// TwinCAT 3 PLC project PLC
// ProgramVersion: 3.1.4023.0
// libraries:
//   Tc2_MC2, * (Beckhoff Automation GmbH)
//   Tc2_Standard, * (Beckhoff Automation GmbH)
//   Tc2_System, * (Beckhoff Automation GmbH)
//   Tc3_MC2_AdvancedHoming, * (Beckhoff Automation GmbH)
//   Tc3_Module, * (Beckhoff Automation GmbH)
// project tree:
//   DUTs/Motion/ E_AxisParameters.TcTLEO, E_EncoderTypeClass.TcDUT, E_HomeSwitchTypeClass.TcDUT, E_HomingRoutines.TcTLEO, E_MotionFunctions.TcDUT, E_MotorTypeClass.TcDUT, E_RestorePosition.TcDUT, ST_AxisConfig.TcDUT, ST_AxisControl.TcDUT, ST_AxisDescription.TcDUT, ST_AxisError.TcDUT, ST_AxisInputs.TcDUT, ST_AxisPersistent.TcDUT, ST_AxisStatus.TcDUT, ST_AxisStruct.TcDUT, ST_GearAxis.TcDUT
//   GVLs/ GVL_APP.TcGVL, GVL.TcGVL
//   / PlcTask.TcTTO
//   POUs/ MAIN.TcPOU
//   POUs/Motion/ FB_Axis.TcPOU
//   POUs/Motion/Homing/ FB_Homing.TcPOU
// real-time tasks:
//   TASK PlcTask: cycle T#10ms, priority 20, ADS port 350
// motion (NC):
//   TASK NC-Task 1 SAF: cycle T#2ms, priority 4, ADS port 501
//   TASK NC-Task 1 SVB: cycle T#10ms, priority 8, ADS port 511
//   AXIS R1_Axis01_X1 (id 1)
//     OtherSettings: AllowMotionCmdToSlave=true
//     encoder EncType=1
//     drive DrvType=5
//       Analog: TorqueSetpointScale=10, ScaleFactorActTorque=0.1
//     controller CtrType=1
//       CtrPara: PriorControlFactor=1
//         Observer: BandWidth=20
//   AXIS R1_Axis02_X2 (id 2)
//     OtherSettings: AllowMotionCmdToSlave=true
//     encoder EncType=1
//     drive DrvType=5
//       Analog: TorqueSetpointScale=10, ScaleFactorActTorque=0.1
//     controller CtrType=1
//       CtrPara: PriorControlFactor=1
//         Observer: BandWidth=20
//   AXIS R1_Axis03_Y (id 3)
//     OtherSettings: AllowMotionCmdToSlave=true
//     encoder EncType=1
//     drive DrvType=5
//       Analog: TorqueSetpointScale=10, ScaleFactorActTorque=0.1
//     controller CtrType=1
//       CtrPara: PriorControlFactor=1
//         Observer: BandWidth=20
//   AXIS R1_Axis04_Z (id 4)
//     OtherSettings: AllowMotionCmdToSlave=true
//     encoder EncType=1
//     drive DrvType=5
//       Analog: TorqueSetpointScale=10, ScaleFactorActTorque=0.1
//     controller CtrType=1
//       CtrPara: PriorControlFactor=1
//         Observer: BandWidth=20
// variable links:
//   PLC/PLC Instance <-> NC-Task 1 SAF/Axes/R1_Axis01_X1
//     PlcTask Inputs/GVL.astAxes[1].Axis.NcToPlc <-> Outputs/ToPlc
//     PlcTask Outputs/GVL.astAxes[1].Axis.PlcToNc <-> Inputs/FromPlc
//   PLC/PLC Instance <-> NC-Task 1 SAF/Axes/R1_Axis02_X2
//     PlcTask Inputs/GVL.astAxes[2].Axis.NcToPlc <-> Outputs/ToPlc
//     PlcTask Outputs/GVL.astAxes[2].Axis.PlcToNc <-> Inputs/FromPlc
//   PLC/PLC Instance <-> NC-Task 1 SAF/Axes/R1_Axis03_Y
//     PlcTask Inputs/GVL.astAxes[3].Axis.NcToPlc <-> Outputs/ToPlc
//     PlcTask Outputs/GVL.astAxes[3].Axis.PlcToNc <-> Inputs/FromPlc
//   PLC/PLC Instance <-> NC-Task 1 SAF/Axes/R1_Axis04_Z
//     PlcTask Inputs/GVL.astAxes[4].Axis.NcToPlc <-> Outputs/ToPlc
//     PlcTask Outputs/GVL.astAxes[4].Axis.PlcToNc <-> Inputs/FromPlc

CONFIGURATION PLC
    RESOURCE PLC ON TwinCAT3
        TASK PlcTask(INTERVAL := T#10ms, PRIORITY := 20);
        PROGRAM MAIN WITH PlcTask : MAIN;
    END_RESOURCE
END_CONFIGURATION

// ---- DUTs/Motion/E_AxisParameters.TcTLEO
{attribute 'qualified_only'}
{attribute 'strict'}
TYPE E_AxisParameters :
(
//PLCopen specific parameters Index-Group 0x4000 + ID
    CommandedPosition := 1, //lreal taken from NcToPlc
    SWLimitForward := 2, //lreal IndexOffset= 16#0001_000E
    SWLimitBackward := 3, //lreal IndexOffset= 16#0001_000D
    EnableLimitForward := 4, //bool IndexOffset= 16#0001_000C
    EnableLimitBackward := 5, //bool IndexOffset= 16#0001_000B
    EnablePositionLagMonitoring := 6, //bool IndexOffset= 16#0002_0010
    MaxPositionLag := 7, //lreal IndexOffset= 16#0002_0012
    AxisMaxVelocity := 8, //lreal IndexOffset= 16#0000_0027
    ActualVelocity := 10, //lreal taken from NcToPlc
    CommandedVelocity := 11, //lreal taken from NcToPlc
    AxisDefaultAcceleration := 12, //lreal IndexOffset= 16#0000_0101
    AxisDefaultDeceleration := 14, //lreal IndexOffset= 16#0000_0102
    AxisDefaultJerk := 16, //lreal IndexOffset= 16#0000_0103

//Beckhoff specific parameters Index-Group 0x4000 + ID
    AxisId := 1000, //lreal IndexOffset= 16#0000_0001
    AxisManualVelocitySlow := 1001, //lreal IndexOffset= 16#0000_0008
    AxisManualVelocityFast := 1002, //lreal IndexOffset= 16#0000_0009
    AxisAccMax := 1004, //lreal IndexOffset= 16#0000_0101
    AxisDecMax := 1005, //lreal IndexOffset= 16#0000_0102
    AxisRapidTraverseVelocity := 1009, //lreal IndexOffset= 16#0000_000A
    AxisVelocityToCam := 1012, //lreal IndexOffset= 16#0000_0006
    AxisVelocityFromCam := 1013, //lreal IndexOffset= 16#0000_0007
    AxisJogIncrementForward := 1014, //lreal IndexOffset= 16#0000_0018
    AxisJogIncrementBackward := 1015, //lreal IndexOffset= 16#0000_0019
    MaxPositionLagFilterTime := 1022, //lreal IndexOffset= 16#0002_0013
    AxisEnPositionRangeMonitoring := 1023, //bool IndexOffset= 16#0000_000F
    AxisPositionRangeWindow := 1024, //lreal IndexOffset= 16#0000_0010
    AxisEnTargetPositionMonitoring:= 1025, //bool IndexOffset= 16#0000_0015
    AxisTargetPositionWindow := 1026, //lreal IndexOffset= 16#0000_0016
    AxisTargetPositionMonitoringTime := 1027, //lreal IndexOffset= 16#0000_0017
    AxisEnInTargetTimeout := 1028, //bool IndexOffset= 16#0000_0029
    AxisInTargetTimeout := 1029, //lreal IndexOffset= 16#0000_002A
    AxisEnMotionMonitoring := 1030, //bool IndexOffset= 16#0000_0011
    AxisMotionMonitoringWindow := 1031, //lreal IndexOffset= 16#0000_0028
    AxisMotionMonitoringTime := 1032, //lreal IndexOffset= 16#0000_0012
    AxisDelayTimeVeloPosition := 1033, //lreal IndexOffset= 16#0000_0104
    AxisEnLoopingDistance := 1034, //bool IndexOffset= 16#0000_0013
    AxisLoopingDistance := 1035, //lreal IndexOffset= 16#0000_0014
    AxisEnBacklashCompensation := 1036, //bool IndexOffset= 16#0000_002B
    AxisBacklash := 1037, //lreal IndexOffset= 16#0000_002C
    AxisEnDataPersistence := 1038, //bool IndexOffset= 16#0000_0030
    AxisRefVeloOnRefOutput := 1039, //lreal IndexOffset= 16#0003_0101
    AxisOverrideType := 1040, //lreal IndexOffset= 16#0000_0105
    //new since 4/2007
    AxisEncoderOffset := 1042, //lreal IndexOffset= 16#0001_0007
    AxisEncoderDirectionInverse := 1043, //bool IndexOffset= 16#0001_0008
    AxisEncoderMask := 1044, //dword IndexOffset= 16#0001_0015
    AxisEncoderModuloValue := 1045, //lreal IndexOffset= 16#0001_0009
    AxisModuloToleranceWindow := 1046, //lreal IndexOffset= 16#0001_001B
    AxisEnablePosCorrection := 1047, //bool IndexOffset= 16#0001_0016
    AxisPosCorrectionFilterTime := 1048, //lreal IndexOffset= 16#0001_0017
    //new since 1/2010
    AxisUnitInterpretation := 1049, //lreal IndexOffset= 16#0000_0026
    AxisMotorDirectionInverse := 1050, //bool  IndexOffset= 16#0003_0006
    //new since 1/2011
    AxisCycleTime := 1051, //lreal IndexOffset= 16#0000_0004
    //new since 5/2011
    AxisFastStopSignalType := 1052, //dword IndexOffset= 16#0000_001E
    AxisFastAcc := 1053, //lreal IndexOffset= 16#0000_010A
    AxisFastDec := 1054, //lreal IndexOffset= 16#0000_010B
    AxisFastJerk := 1055, //lreal IndexOffset= 16#0000_010C
    // new since 1/2012 *)
    AxisEncoderScalingNumerator := 1056, //lreal IndexOffset= 16#0001_0023 - available in Tc3
    AxisEncoderScalingDenominator := 1057, //lreal IndexOffset= 16#0001_0024 - available in Tc3
    (* new since 7/2016 *)
    AxisVeloJumpFactor := 1060, //lreal IndexOffset= 16#0000_0106
    AxisToleranceBallAuxAxis := 1061, //lreal IndexOffset= 16#0000_0108
    AxisMaxPositionDeviationAuxAxis := 1062, //lreal IndexOffset= 16#0000_0109
    AxisErrorPropagationMode := 1063, //dword IndexOffset= 16#0000_001A
    AxisErrorPropagationDelay := 1064, //lreal IndexOffset= 16#0000_001B
    AxisCoupleSlaveToActualValues := 1065, //bool IndexOffset= 16#0000_001C
    AxisAllowMotionCmdToSlaveAxis := 1066, //bool IndexOffset= 16#0000_0020
    AxisAllowMotionCmdToExtSetAxis := 1067, //bool IndexOffset= 16#0000_0021
    AxisEncoderSubMask := 1068, //dword IndexOffset= 16#0001_0108
    AxisEncoderReferenceSystem := 1069, //dword IndexOffset= 16#0001_0019
    AxisEncoderPositionFilterPT1 := 1070, //lreal IndexOffset= 16#0001_0010
    AxisEncoderVelocityFilterPT1 := 1071, //lreal IndexOffset= 16#0001_0011
    AxisEncoderAccelerationFilterPT1 := 1072, //lreal IndexOffset= 16#0001_0012
    AxisEncoderMode := 1073, //dword IndexOffset= 16#0001_000A
    AxisEncoderHomingInvDirCamSearch := 1074, //bool IndexOffset= 16#0001_0101
    AxisEncoderHomingInvDirSyncSearch := 1075, //bool IndexOffset= 16#0001_0102
    AxisEncoderHomingCalibValue := 1076, //lreal IndexOffset= 16#0001_0103
    AxisEncoderReferenceMode := 1077, //dword IndexOffset= 16#0001_0107
    AxisRefVeloOutputRatio := 1078, //lreal IndexOffset= 16#0003_0102
    AxisDrivePositionOutputScaling := 1079, //lreal IndexOffset= 16#0003_0109
    AxisDriveVelocityOutputScaling := 1080, //lreal IndexOffset= 16#0003_0105
    AxisDriveVelocityOutputDelay := 1081, //lreal IndexOffset= 16#0003_010D
    AxisDriveMinOutputLimitation := 1082, //lreal IndexOffset= 16#0003_000B
    AxisDriveMaxOutputLimitation := 1083, //lreal IndexOffset= 16#0003_000C
    AxisTorqueInputScaling := 1084, //lreal IndexOffset= 16#0003_0031 - available in Tc3
    AxisTorqueInputFilterPT1 := 1085, //lreal IndexOffset= 16#0003_0032 - available in Tc3
    AxisTorqueDerivationInputFilterPT1 := 1086, //lreal IndexOffset= 16#0003_0033 - available in Tc3
    AxisTorqueOutputScaling := 1087, //lreal IndexOffset= 16#0003_010B
    AxisTorqueOutputDelay := 1088, //lreal IndexOffset= 16#0003_010F
    AxisAccelerationOutputScaling := 1089, //lreal IndexOffset= 16#0003_010A
    AxisAccelerationOutputDelay := 1090, //lreal IndexOffset= 16#0003_010E
    AxisDrivePositionOutputSmoothFilterType := 1091, //dword IndexOffset= 16#0003_0110
    AxisDrivePositionOutputSmoothFilterTime := 1092, //lreal IndexOffset= 16#0003_0111
    AxisDrivePositionOutputSmoothFilterOrder := 1093, //dword IndexOffset= 16#0003_0112
    AxisDriveMode := 1094, //dword IndexOffset= 16#0003_000A
    AxisDriftCompensationOffset := 1095, //lreal IndexOffset= 16#0003_0104
    AxisPositionControlKv := 1096, //lreal IndexOffset= 16#0002_0102
    AxisCtrlVelocityPreCtrlWeight := 1097, //lreal IndexOffset= 16#0002_000B
    AxisControllerMode := 1098, //dword IndexOffset= 16#0002_000A
    AxisCtrlAutoOffset := 1099, //bool IndexOffset= 16#0002_0110
    AxisCtrlAutoOffsetTimer := 1100, //lreal IndexOffset= 16#0002_0115
    AxisCtrlAutoOffsetLimit := 1101, //lreal IndexOffset= 16#0002_0114
    AxisSlaveCouplingControlKcp := 1102, //lreal IndexOffset= 16#0002_010F
    AxisCtrlOutputLimit := 1103, //lreal IndexOffset= 16#0002_0100

//Beckhoff specific axis status information - READ ONLY Index-Group 0x4100 + ID
    AxisTargetPosition := 2000, //lreal IndexOffset= 16#0000_0013
    AxisRemainingTimeToGo := 2001, //lreal IndexOffset= 16#0000_0014
    AxisRemainingDistanceToGo := 2002, //lreal IndexOffset= 16#0000_0022, 16#0000_0042

//Beckhoff specific axis functions
    //read/write gear ratio of a slave
    AxisGearRatio := 3000, //lreal read: IndexGroup=0x4100+ID, IdxOffset=16#0000_0022,
                                 //write:IndexGroup=0x4200+ID, IdxOffset=16#0000_0042

//Beckhoff specific other parameters
    //new since 1/2011
    NcSafCycleTime := 4000, //lreal IndexOffset= 16#0000_0010
    NcSvbCycleTime := 4001 //lreal IndexOffset= 16#0000_0012

);
END_TYPE

// ---- DUTs/Motion/E_EncoderTypeClass.TcDUT
TYPE E_EncoderTypeClass :
(
    eNoEncoder := 0,
    eIncrementalEncoder := 1,
    eAbsoluteEncoder := 2
) := eNoEncoder;
END_TYPE

// ---- DUTs/Motion/E_HomeSwitchTypeClass.TcDUT
TYPE E_HomeSwitchTypeClass:
(
    eNoSwitch := 0, //no physical switch for homing present
    eHomeSwitchPresent := 1, //dedicated homing switch present
    eUseBwdLimit := 2, //Bwd limit switch is used as a homing switch
    eUseFwdLimit := 3 //Fwd limit switch is used as a homing switch
) := eNoSwitch;
END_TYPE

// ---- DUTs/Motion/E_HomingRoutines.TcTLEO
{attribute 'qualified_only'}
{attribute 'strict'}
TYPE E_HomingRoutines :
(
    eNoHoming := 0,

    //0X: LIMIT Switch
    //Home to bBwdLimit, record position on first approach
    eHomeToLimit_Bwd := 1,
    //Home to bFwdLimit, record position on first approach
    eHomeToLimit_Fwd := 2,
    //Find bBwdLimit (using towardsCam speed), then reverse direction looking FOR falling edge (using fromCam speed)
    //eHomeToLimit_Bwd_2Speeds := 3,
    //Find bFwdLimit (using towardsCam speed), then reverse direction looking for falling edge (using fromCam speed)
    //eHomeToLimit_Fwd_2Speeds := 4,

    //1X: Home Sensor
    //Home to bHome in Bwd direction (will reverse direction if limit hit), record position on first approach
    eHomeToRef_Bwd := 11,
    //Home to bHome in Fwd direction (will reverse direction if limit hit), record position on first approach
    eHomeToRef_Fwd := 12,
    //Find bHome in Bwd direction (using towardsCam speed) then reverse direction looking for falling edge (using fromCam speed), will reverse direction if limit hit
    //eHomeToRef_Bwd_2Speeds := 13,
    //Find bHome in Fwd direction (using towardsCam speed) then reverse direction looking for falling edge (using fromCam speed), will reverse direction if limit hit
    //eHomeToRef_Fwd_2Speeds := 14,

    //2X: Enc Pulse
    //Home to EncRefPulse in Bwd direction (used for single turn rotary axis without limit switches)
    eHomeToEncPulse_Bwd := 21,
    //Home to EncRefPulse in Fwd direction (used for single turn rotary axis without limit switches)
    eHomeToEncPulse_Fwd := 22,
    //Home to EncRefPulse via bBwdLimit (using towardsCam speed), then reverse direction looking for falling edge on ref pulse (using fromCam speed)
    eHomeToEncPulse_viaBwdLimit := 23,
    //Home to EncRefPulse via bFwdLimit (using towardsCam speed), then reverse direction looking for falling edge on ref pulse (using fromCam speed)
    eHomeToEncPulse_viaFwdLimit := 24,

    //9X: Software
    eHomeDirect := 90 //Set position directly to fHomePosition
) := eNoHoming;
END_TYPE

// ---- DUTs/Motion/E_MotionFunctions.TcDUT
{attribute 'qualified_only'}
{attribute 'strict'}
TYPE E_MotionFunctions :
(
    eMoveAbsolute 		:= 0,
    eMoveRelative 		:= 1,
    eJog 				:= 2, //Continous moving in the direction specified by bJogFwd or bJogBwd as long as one is high. Will stop if bExecute goes high. Generally not called by an external control system.
    eMoveVelocity 		:= 3, //Continous moving at a set velocity once bExecute goes high
    eMoveModulo 		:= 4, //Move for 360 deg rotation, see Beckhoff docs
    eGearIn 			:= 5, //Gears in this axis to be the slave of the axis specified in masterAxis with the ratio specified in there
    eGearOut 			:= 6, //Removes gearing set in the above command
    eGearInMultiMaster 	:= 7, //Gears in this axis to be the slave of the axis specified in stMultiMasterAxis with the ratio specified
    eHome 				:= 10, //Run the homing routine for the axis
    eWriteParameter 	:= 50 //Writes the set value to the set parameter once bExecute goes high
) 	:= eJog; //Jog is the default behaviour of the axis.
END_TYPE

// ---- DUTs/Motion/E_MotorTypeClass.TcDUT
TYPE E_MotorTypeClass :
(
    eVirtualMotor := 0, //Axis is Virtual
    eStepperMotor := 1, //Axis based on a stepper motor
    eDcMotor := 2, //Axis based on a brushed DC motor
    eBldcMotor := 3, //Axis based on a BLDC motor
    eAsyncMotor := 4, //Axis based on a three phase asynchronous motor
    eSyncMotor := 5 //Axis based on a three phase synchronous motor
) := eVirtualMotor;
END_TYPE

// ---- DUTs/Motion/E_RestorePosition.TcDUT
{attribute 'qualified_only'}
{attribute 'strict'}
TYPE E_RestorePosition :
(
    eDontRestore :=0,
    eRestoreWithoutHome := 1 //Redefined the position of the axis to that when the power was lost
);
END_TYPE

// ---- DUTs/Motion/ST_AxisConfig.TcDUT
(*These are axis parameters that are set up during commissioning and
in theory don't neeed to be change as part of daily moving of axes.
For instance they may be changed due to poor parameter selection
or change of instrument configuration.*)
TYPE ST_AxisConfig :
STRUCT
    //Axis Parameters
    fOverride: LREAL := 100; //Controller override %, used a global scale for an axis in terms of velocity. Generally set to 100%.
    fHomePosition: LREAL := 0; //The position that the axis should be set to once homing is completed
    fHomeFinishDistance: LREAL := 0; //Distrance that the axis should move back into the working zone after homing is finished
    eHomeSeq: E_HomingRoutines; //Homing sequence to perform
    eRestorePosition: E_RestorePosition; //Restore position of incremental axis after loss of power to the CPU, 0=don't restore, 1=restore but don't home

    //Read and Write parameters
    eAxisParameters: E_AxisParameters; //Enumeration of axis parameters
    fWriteAxisParameter: LREAL; //The value to be writen to eAxisParameterNumber
    fReadAxisParameter: LREAL; //Read the current value of the selected eAxisParameterNumber
    bReadAxisParameterValid: BOOL; //Is the current data thats been read valid value

    //Single master axis parameters
    stMasterAxis: ST_GearAxis; //A reference to the axis that this is a slave of
    afSlaveAxisRatio: ARRAY [1..GVL_APP.nAXIS_NUM] OF LREAL; //The gearing between this axis as a master and any slaves. e.g. if this is a 1 to 1 master of axis 2 this will be [0, 1, 0 ...]

    //Multi master axis parameters
    astMultiMasterAxis: ARRAY [1..4] OF ST_GearAxis;
    astMultiMasterAxisLatched: ARRAY [1..4] OF ST_GearAxis; //A kind of readback since one doesn't exist in AXIS_REF
    afMultiSlaveAxisRatio: ARRAY [1..GVL_APP.nAXIS_NUM] OF LREAL;

    // Read only MC parameters
    bReadMcParametersValid: BOOL:= FALSE;
    bReadMcParametersError: BOOL:= FALSE;
    fVelocityDefaultSlow: LREAL; //Read only - AxisVeloManSlow
    fVelocityDefaultFast: LREAL; //Read only - AxisVeloManFast
    fHomingVelToCam: LREAL; //Read only - AxisCalibrationVelocityForward
    fHomingVelFromCam: LREAL; //Read only - AxisCalibrationVelocityBackward
    fVeloMax: LREAL; //Read only - fVeloMax
    fDefaultAcc: LREAL; //Read only - AxisAcc
    fDefaultDec: LREAL; //Read only - AxisDec
    bEnMinSoftPosLimit: BOOL; //Read only
    fMinSoftPosLimit: LREAL; //Read only
    bEnMaxSoftPosLimit: BOOL; //Read only
    fMaxSoftPosLimit: LREAL; //Read only
    bEnPositionLagMonitoring: BOOL; //Read only
    fMaxPosLagValue: LREAL; //Read only
    bEnTargetPositionMonitoring: BOOL; //Read only
    fTargetPositionWindow: LREAL; //Read only
END_STRUCT
END_TYPE

// ---- DUTs/Motion/ST_AxisControl.TcDUT
(*These are parameters that are used to initiate axis movements
They are commands that are commonly used commands*)
TYPE ST_AxisControl :
STRUCT
    //Actions from controls system
    bExecute		: 	BOOL; //Rising edge to execute some motion FB's
    bReset			: 	BOOL; //Reset axis from Error state
    bStop			: 	BOOL;
    bHalt			: 	BOOL;
    bEnable			: 	BOOL; //Enable axis drive
    bJogFwd			: 	BOOL;
    bJogBwd			: 	BOOL;
    eCommand		: 	E_MotionFunctions;
    fVelocity		: 	LREAL; //Velocity must be specified, no default used
    fAcceleration	: 	LREAL; //Not all FBs use, 0 is NC default
    fDeceleration	: 	LREAL;
    fPosition		: 	LREAL; //The position to move to for an absolute move and the amount to move in a relative move
END_STRUCT
END_TYPE

// ---- DUTs/Motion/ST_AxisDescription.TcDUT
TYPE ST_AxisDescription :
STRUCT
    sAxisName : STRING(nMAX_AXIS_NAME);
    nUnit: BYTE; //Code for the axis base unit (like m or degree)
    nPrefix: BYTE; //Exponent defining unit prefix, e.g. 3 for k(kilo)
    bIsPseudoAxis: BOOL; //Axis is a non-standard axis with application-specific handling
    eEncoderType: E_EncoderTypeClass;
    eHomeSwitchType: E_HomeSwitchTypeClass;
    eMotorType: E_MotorTypeClass;
END_STRUCT
END_TYPE

// ---- DUTs/Motion/ST_AxisError.TcDUT
TYPE ST_AxisError:
STRUCT
//PLCopen function block errors
    nPowerErrorID : UDINT;
    nMoveAbsoluteErrorID : UDINT;
    nMoveRelativeErrorID : UDINT;
    nMoveVelocityErrorID : UDINT;
    nMoveModuloErrorID : UDINT;
    nJogErrorID : UDINT;
    nHomeErrorID : UDINT;
    nHaltErrorID : UDINT;
    nResetErrorID : UDINT;
    nStopErrorID : UDINT;
    nGearInErrorID : UDINT;
    nGearInMultiMasterErrorID : UDINT;
    nGearOutErrorID : UDINT;
    fbWriteParameterErrorId : UDINT;
    fbReadParameterErrorId : UDINT;
//Error from the NC
    nNCErrorID : UDINT;
END_STRUCT
END_TYPE

// ---- DUTs/Motion/ST_AxisInputs.TcDUT
TYPE ST_AxisInputs :
STRUCT
    bLimitFwd AT %I*: BOOL;
    bLimitBwd AT %I*: BOOL;
    bHomeSensor AT %I*: BOOL; //Reference siganl for homing
END_STRUCT
END_TYPE

// ---- DUTs/Motion/ST_AxisPersistent.TcDUT
TYPE ST_AxisPersistent :
STRUCT
    //Settings for restoring positions on power off
    fPositionAtShutdown: LREAL; //The position that the axis was at when CPU shut down
    bMovingAtShutdown: BOOL; //True if the axis was moving at shutdown, False otherwise
END_STRUCT
END_TYPE

// ---- DUTs/Motion/ST_AxisStatus.TcDUT
TYPE ST_AxisStatus :
STRUCT
    //Outputs & Status
    bEnabled: BOOL; //Axis drive enabled
    bCommandAborted: BOOL; //Command aborted output of the eCommand function blocks
    bBusy: BOOL; //Axis busy (eCommand function block is active)
    bDone: BOOL; //Last eCommand function block executed successfully;
    //bDone will also be set with the InGear and InVelocity outputs
    //When InVelocity is set, fbMoveVelocity is still acitve, which is reflected by the bBusy status
    bHomed: BOOL; //Axis homed
    bMoving: BOOL; //Moving state from the NC
    bFwEnabled: BOOL; //Positive movement of axis is enabled/disabled
    bBwEnabled: BOOL; //Negative movement of axis is enabled/disabled
    bGeared: BOOL; //Axis is an active slave
    bCoupledGear1: BOOL;
    bCoupledGear2: BOOL;
    bCoupledGear3: BOOL;
    bCoupledGear4: BOOL;
    fActPosition: LREAL; //Actual position value
    fActVelocity: LREAL; //Actual velocity
    bError: BOOL; //Motion function block has produced error (NC drive not necessarily in error state)
    nErrorID: UDINT; //Last motion function block errorID or NC errorID
END_STRUCT
END_TYPE

// ---- DUTs/Motion/ST_AxisStruct.TcDUT
TYPE ST_AxisStruct :
STRUCT
    stControl	:	ST_AxisControl;
    stStatus	: 	ST_AxisStatus;
    stConfig	: 	ST_AxisConfig;
    stError		: 	ST_AxisError;
    stInputs	: 	ST_AxisInputs;
    Axis		: 	tc2_mc2.AXIS_REF; //The NC axis link to the hardware that is controlling
END_STRUCT
END_TYPE

// ---- DUTs/Motion/ST_GearAxis.TcDUT
TYPE ST_GearAxis :
STRUCT
    nIndex: UINT := 1; //Index of the master axis
    fRatio: LREAL := 0; //Gearing ratio between master axis and this one
END_STRUCT
END_TYPE

// ---- GVLs/GVL_APP.TcGVL
{attribute 'qualified_only'}
VAR_GLOBAL
END_VAR

VAR_GLOBAL CONSTANT
	nAXIS_NUM			: 	UINT := 4;
END_VAR

// ---- GVLs/GVL.TcGVL
VAR_GLOBAL
    astAxes				: 	ARRAY [1..GVL_APP.nAXIS_NUM] OF ST_AxisStruct; //Global array of ST_AxisStruct for holding axis parameters and controls
    iAxis				: 	UINT; //Index for for loops while going through axes
END_VAR

VAR_GLOBAL CONSTANT
    nMAX_AXIS_NAME		: 	UINT := 32;
END_VAR

VAR_GLOBAL PERSISTENT
    astAxesPersistent	: 	ARRAY [1..GVL_APP.nAXIS_NUM] OF ST_AxisPersistent;
END_VAR

// ---- POUs/MAIN.TcPOU
PROGRAM MAIN
VAR
	FB_Axis_X1 	: 	FB_Axis;
	st_Axis_X1	: 	ST_AxisStruct;
	
//	FB_Axis_X2 	: 	FB_Axis;
//	FB_Axis_Y 	: 	FB_Axis;
//	FB_Axis_Z 	: 	FB_Axis;
END_VAR

//st_Axis_X1.stControl.bEnable := TRUE;
st_Axis_X1.stStatus.bFwEnabled := TRUE;
st_Axis_X1.stStatus.bBwEnabled := TRUE;
FB_Axis_X1(stAxisStruct:= st_Axis_X1 );

END_PROGRAM

// ---- POUs/Motion/FB_Axis.TcPOU
//Function block to run a virtual drive with Nc
FUNCTION_BLOCK FB_Axis
VAR
    sVersion						: 	STRING := '1.0.4';
END_VAR

VAR CONSTANT
    nMULTI_MASTER_MAX_AXES			: 	UINT := 4;
    //Kept static as numerator is LREAL and consistent with multigearing
    nRATIO_DENOMINATOR_DEFAULT		: 	UINT := 1;
    //By default 0 as represents no existing gearing
    nNO_GEARING						: 	UINT := 0;
END_VAR

VAR_IN_OUT
    stAxisStruct					: 	ST_AxisStruct;
END_VAR

VAR
    nAxisIndex						: 	UINT;
    nMultiMastersAxesIndex			: 	UINT;
    nSlaveAxesIndex					: 	UINT;
    bWaitForStoppingAfterLimitHit 	: 	BOOL := FALSE;
    fbRemovePowerTimer				: 	TOF;
    stMasterAxis					: 	ST_GearAxis := (nIndex := 1, fRatio := 0);
    fbReset							: 	MC_Reset;
    fbPower							: 	MC_Power;
    fbStop							: 	MC_Stop;
    fbHalt							: 	MC_Halt;
    fbJog							: 	MC_Jog;
    fbMoveAbsolute					: 	MC_MoveAbsolute;
    fbMoveVelocity					: 	MC_MoveVelocity;
    fbMoveRelative					: 	MC_MoveRelative;
    fbMoveModulo					: 	MC_MoveModulo;
    fbGearIn						: 	MC_GearIn;
    fbGearOut						: 	MC_GearOut;
    fbGearInMultiMaster				: 	MC_GearInMultiMaster;
    fbHome							: 	FB_Homing;
    fbExecuteRiseEdge				: 	R_TRIG;
    fbJogRiseEdge					: 	R_TRIG;
    fbStopRiseEdge					: 	R_TRIG;
    fbHaltRiseEdge					: 	R_TRIG;
    fbResetRiseEdge: R_TRIG;
    fbStopFinishedRiseEdge: R_TRIG;
    fbHaltFinishedRiseEdge: R_TRIG;
    fbResetFinishedRiseEdge: R_TRIG;
    fbCommandAbortedRiseEdge: R_TRIG;
    fbDoneRiseEdge: R_TRIG;
    fbWriteParameter: MC_WriteParameter;
    fbReadParameter: MC_ReadParameter;

    // Used in/for actReadMcParameters
    bReadValid: BOOL := FALSE;
    fbReadAxisVeloManSlow: MC_ReadParameter;
    fbReadAxisVeloManFast: MC_ReadParameter;
    fbReadHomingVelToCam: MC_ReadParameter;
    fbReadHomingVelFromCam: MC_ReadParameter;
    fbReadAxisVeloMax: MC_ReadParameter;
    fbReadAxisAcc: MC_ReadParameter;
    fbReadAxisDec: MC_ReadParameter;
    fbReadEnMinSoftPosLimit: MC_ReadParameter;
    fbReadEnMaxSoftPosLimit: MC_ReadParameter;
    fbReadMinSoftPosLimit: MC_ReadParameter;
    fbReadMaxSoftPosLimit: MC_ReadParameter;
    fbReadEnPositionLagMonitoring: MC_ReadParameter;
    fbReadAxisMaxPosLagValue: MC_ReadParameter;
    fbReadEnTargetPositionMonitoring: MC_ReadParameter;
    fbReadTargetPositionWindow: MC_ReadParameter;

    bDoneEdge: BOOL; // helper variable for the detection of a rising edge of the done output of any motion FBs
    bCommandAbortedEdge: BOOL; // helper variable for the detection of a rising edge of the commandAborted output of any motion FBs
    bBusy: BOOL; // helper variable for a logical OR of the busy output of all motion FBs
END_VAR

bBusy := FALSE;

stAxisStruct.Axis.ReadStatus();

actReadMcParameters();

//Call of all MC Instances and set all Executes to FALSE
fbPower(Axis := stAxisStruct.Axis);
fbPower.Enable := FALSE;

fbReset(Axis := stAxisStruct.Axis);
fbReset.Execute := FALSE;
bBusy:= bBusy OR fbReset.Busy;

fbStop(Axis := stAxisStruct.Axis);
fbStop.Execute := FALSE;
bBusy:= bBusy OR fbStop.Busy;

fbHalt(Axis := stAxisStruct.Axis);
fbHalt.Execute := FALSE;
bBusy:= bBusy OR fbHalt.Busy;

fbJog(Axis := stAxisStruct.Axis);
bBusy:= bBusy OR fbJog.Busy;

fbHome(Axis := stAxisStruct.Axis,
bLimitBwd := stAxisStruct.stInputs.bLimitBwd,
bLimitFwd := stAxisStruct.stInputs.bLimitFwd,
bHomeSensor := stAxisStruct.stInputs.bHomeSensor);
fbHome.bExecute := FALSE;
bBusy:= bBusy OR fbHome.bBusy;

fbMoveAbsolute(Axis := stAxisStruct.Axis);
fbMoveAbsolute.Execute := FALSE;
bBusy:= bBusy OR fbMoveAbsolute.Busy;

fbMoveRelative(Axis := stAxisStruct.Axis);
fbMoveRelative.Execute := FALSE;
bBusy:= bBusy OR fbReset.Busy;

fbMoveVelocity(Axis := stAxisStruct.Axis);
fbMoveVelocity.Execute := FALSE;
bBusy:= bBusy OR fbMoveRelative.Busy;

fbMoveModulo(Axis := stAxisStruct.Axis);
fbMoveModulo.Execute := FALSE;
bBusy:= bBusy OR fbMoveModulo.Busy;

fbGearin(Slave := stAxisStruct.Axis, Master := GVL.astAxes[stMasterAxis.nIndex].Axis);
fbGearIn.Execute := FALSE;
bBusy:= bBusy OR fbGearin.Busy;

fbGearInMultiMaster(Slave := stAxisStruct.Axis,
    Master1 := GVL.astAxes[stAxisStruct.stConfig.astMultiMasterAxisLatched[1].nIndex].Axis,
    Master2 := GVL.astAxes[stAxisStruct.stConfig.astMultiMasterAxisLatched[2].nIndex].Axis,
    Master3 := GVL.astAxes[stAxisStruct.stConfig.astMultiMasterAxisLatched[3].nIndex].Axis,
    Master4 := GVL.astAxes[stAxisStruct.stConfig.astMultiMasterAxisLatched[4].nIndex].Axis);
bBusy:= bBusy OR fbGearInMultiMaster.Busy;

fbGearOut(Slave := stAxisStruct.Axis);
fbGearOut.Execute := FALSE;
bBusy:= bBusy OR fbGearOut.Busy;

fbWriteParameter(Axis := stAxisStruct.Axis);
fbWriteParameter.Execute := FALSE;
bBusy:= bBusy OR fbWriteParameter.Busy;

//Read parameter continuously
fbReadParameter(
    Axis := stAxisStruct.Axis,
    Enable := TRUE,
    ParameterNumber := stAxisStruct.stconfig.eAxisParameters,
    ReadMode := READMODE_CYCLIC);
//do no evaluate fbReadParameter.busy, since this is continuously TRUE

IF NOT fbReadParameter.Error THEN
    stAxisStruct.stConfig.bReadAxisParameterValid := fbReadParameter.Valid;
    stAxisStruct.stconfig.fReadAxisParameter := fbReadParameter.Value;
END_IF

//Read parameter continuously
fbReadParameter(
    Axis := stAxisStruct.Axis,
    Enable := TRUE,
    ParameterNumber := stAxisStruct.stconfig.eAxisParameters,
    ReadMode := READMODE_CYCLIC);

IF NOT fbReadParameter.Error THEN
    stAxisStruct.stConfig.bReadAxisParameterValid := fbReadParameter.Valid;
    stAxisStruct.stconfig.fReadAxisParameter := fbReadParameter.Value;
END_IF

//Linking the limit swtiches
stAxisStruct.stStatus.bFwEnabled := stAxisStruct.stInputs.bLimitFwd;
stAxisStruct.stStatus.bBwEnabled := stAxisStruct.stInputs.bLimitBwd;

FOR nAxisIndex := 1 TO GVL_APP.nAXIS_NUM DO
    IF (stAxisStruct.stConfig.afMultiSlaveAxisRatio[nAxisIndex] <> 0) THEN
        stAxisStruct.stStatus.bFwEnabled := stAxisStruct.stStatus.bFwEnabled AND SEL(stAxisStruct.stConfig.afMultiSlaveAxisRatio[nAxisIndex] > 0, GVL.astAxes[nAxisIndex].stStatus.bBwEnabled, GVL.astAxes[nAxisIndex].stStatus.bFwEnabled);
        stAxisStruct.stStatus.bBwEnabled := stAxisStruct.stStatus.bBwEnabled AND SEL(stAxisStruct.stConfig.afMultiSlaveAxisRatio[nAxisIndex] > 0, GVL.astAxes[nAxisIndex].stStatus.bFwEnabled, GVL.astAxes[nAxisIndex].stStatus.bBwEnabled);
    END_IF
END_FOR

//Timer for keeping power on after limit switch hit, needed for homing routines - if power is lost routines are aborted
fbRemovePowerTimer(IN := stAxisStruct.stInputs.bLimitFwd AND stAxisStruct.stInputs.bLimitBwd, PT := T#100MS);
IF fbHome.bBusy AND (fbRemovePowerTimer.Q OR stAxisStruct.Axis.NcToPlc.AxisState=5) THEN //5=PHASE_ACCNEG
    bWaitForStoppingAfterLimitHit := TRUE;
ELSE
    bWaitForStoppingAfterLimitHit := FALSE;
END_IF

//Power
fbPower.Enable 					:= 	TRUE; //stAxisStruct.stControl.bEnable;
fbPower.Enable_Positive 		:= 	TRUE; //stAxisStruct.stStatus.bFwEnabled OR bWaitForStoppingAfterLimitHit;
fbPower.Enable_Negative 		:= 	TRUE; //stAxisStruct.stStatus.bBwEnabled OR bWaitForStoppingAfterLimitHit;
fbPower.Override 				:= 	100.0; //stAxisStruct.stConfig.fOverride;
stAxisStruct.stStatus.bEnabled	:= 	fbPower.Status;

//Stop
fbStop.Execute := stAxisStruct.stControl.bStop;
fbHalt.Deceleration := stAxisStruct.stControl.fDeceleration;

//Halt
fbHalt.Execute := stAxisStruct.stControl.bHalt;
fbHalt.Deceleration := stAxisStruct.stControl.fDeceleration;

//Reset only if axis is in error state
IF stAxisStruct.stStatus.bError THEN
    fbReset.Execute := stAxisStruct.stControl.bReset;
ELSE
    stAxisStruct.stControl.bReset := FALSE;
END_IF

//Motion Functions
CASE stAxisStruct.stControl.eCommand OF
    E_MotionFunctions.eMoveAbsolute:
        fbMoveAbsolute.Execute := stAxisStruct.stControl.bExecute;
        fbMoveAbsolute.Position := stAxisStruct.stControl.fPosition;
        fbMoveAbsolute.Velocity := ABS(stAxisStruct.stControl.fVelocity);
        fbMoveAbsolute.Acceleration := stAxisStruct.stControl.fAcceleration;
        fbMoveAbsolute.Deceleration := stAxisStruct.stControl.fDeceleration;
        bDoneEdge := fbMoveAbsolute.Done;
        bCommandAbortedEdge := fbMoveAbsolute.CommandAborted;

    E_MotionFunctions.eMoveRelative:
        fbMoveRelative.Execute := stAxisStruct.stControl.bExecute;
        fbMoveRelative.Distance := stAxisStruct.stControl.fPosition;
        fbMoveRelative.Velocity := ABS(stAxisStruct.stControl.fVelocity);
        fbMoveRelative.Acceleration := stAxisStruct.stControl.fAcceleration;
        fbMoveRelative.Deceleration := stAxisStruct.stControl.fDeceleration;
        bDoneEdge := fbMoveRelative.Done;
        bCommandAbortedEdge := fbMoveRelative.CommandAborted;

    E_MotionFunctions.eJog:
        fbJog.JogForward := stAxisStruct.stControl.bJogFwd AND NOT (stAxisStruct.stControl.bExecute OR stAxisStruct.stStatus.bError);
        fbJog.JogBackwards := stAxisStruct.stControl.bJogBwd AND NOT (stAxisStruct.stControl.bExecute OR stAxisStruct.stStatus.bError);
        fbJog.Mode := 0;
        fbJog.Velocity := stAxisStruct.stControl.fVelocity;
        fbJog.Acceleration := stAxisStruct.stControl.fAcceleration;
        fbJog.Deceleration := stAxisStruct.stControl.fDeceleration;
        bDoneEdge := fbJog.Done;
        bCommandAbortedEdge := fbJog.CommandAborted;

    E_MotionFunctions.eMoveVelocity:
        fbMoveVelocity.Execute := stAxisStruct.stControl.bExecute;
        fbMoveVelocity.Velocity := ABS(stAxisStruct.stControl.fVelocity);
        fbMoveVelocity.Acceleration := stAxisStruct.stControl.fAcceleration;
        fbMoveVelocity.Deceleration := stAxisStruct.stControl.fDeceleration;
        fbMoveVelocity.Direction := SEL(stAxisStruct.stControl.fVelocity < 0, MC_Positive_Direction, MC_Negative_Direction);
        bCommandAbortedEdge := fbMoveVelocity.CommandAborted;

    E_MotionFunctions.eMoveModulo:
        fbMoveModulo.Execute := stAxisStruct.stControl.bExecute;
        fbMoveModulo.Position := stAxisStruct.stControl.fPosition;
        fbMoveModulo.Velocity := ABS(stAxisStruct.stControl.fVelocity);
        fbMoveModulo.Acceleration := stAxisStruct.stControl.fAcceleration;
        fbMoveModulo.Deceleration := stAxisStruct.stControl.fDeceleration;
        bDoneEdge := fbMoveModulo.Done;
        bCommandAbortedEdge := fbMoveModulo.CommandAborted;

    E_MotionFunctions.eGearIn:
        fbGearIn.Execute := stAxisStruct.stControl.bExecute;
        fbGearIn.RatioNumerator := stMasterAxis.fRatio;
        fbGearIn.RatioDenominator := nRATIO_DENOMINATOR_DEFAULT;
        bCommandAbortedEdge := fbGearIn.CommandAborted;

        IF NOT fbGearIn.InGear THEN
            stMasterAxis.nIndex := stAxisStruct.stConfig.stMasterAxis.nIndex;
            stMasterAxis.fRatio := stAxisStruct.stConfig.stMasterAxis.fRatio;
        END_IF

        //Confirm slaves have no gearing before attempting to gear in
         IF fbGearIn.InGear AND (GVL.astAxes[stMasterAxis.nIndex].stConfig.afSlaveAxisRatio[GVL.iAxis] = nNO_GEARING) THEN
            GVL.astAxes[stMasterAxis.nIndex].stConfig.afSlaveAxisRatio[GVL.iAxis] := stMasterAxis.fRatio;
        END_IF

    E_MotionFunctions.eGearInMultiMaster:
        bCommandAbortedEdge := fbGearInMultiMaster.CommandAborted;

        IF stAxisStruct.stControl.bExecute AND NOT stAxisStruct.Axis.Status.Coupled THEN
            //Latch master references
            FOR nMultiMastersAxesIndex := 1 TO nMULTI_MASTER_MAX_AXES DO
                IF stAxisStruct.stConfig.astMultiMasterAxis[nMultiMastersAxesIndex].nIndex > 0 AND stAxisStruct.stConfig.astMultiMasterAxis[nMultiMastersAxesIndex].nIndex <= GVL_APP.nAXIS_NUM THEN
                    stAxisStruct.stConfig.astMultiMasterAxisLatched[nMultiMastersAxesIndex].nIndex := stAxisStruct.stConfig.astMultiMasterAxis[nMultiMastersAxesIndex].nIndex;
                END_IF
            END_FOR
            //Latch gear ratios
            FOR nMultiMastersAxesIndex := 1 TO nMULTI_MASTER_MAX_AXES DO
                stAxisStruct.stConfig.astMultiMasterAxisLatched[nMultiMastersAxesIndex].fRatio := stAxisStruct.stConfig.astMultiMasterAxis[nMultiMastersAxesIndex].fRatio;
            END_FOR
            //Transfer gear ratios to FB
            fbGearInMultiMaster.GearRatio1 := stAxisStruct.stConfig.astMultiMasterAxisLatched[1].fRatio;
            fbGearInMultiMaster.GearRatio2 := stAxisStruct.stConfig.astMultiMasterAxisLatched[2].fRatio;
            fbGearInMultiMaster.GearRatio3 := stAxisStruct.stConfig.astMultiMasterAxisLatched[3].fRatio;
            fbGearInMultiMaster.GearRatio4 := stAxisStruct.stConfig.astMultiMasterAxisLatched[4].fRatio;
            fbGearInMultiMaster.Enable := stAxisStruct.stControl.bExecute;
        END_IF

        IF fbGearInMultiMaster.Error THEN
            fbGearInMultiMaster.Enable := FALSE;
        END_IF

    E_MotionFunctions.eGearOut:
        fbGearOut.Execute := stAxisStruct.stControl.bExecute;
        fbGearInMultiMaster.Enable := FALSE;
        bDoneEdge := fbGearOut.Done;

        IF fbGearOut.Done THEN
            //Clear slave ratio from master axis slave array
            GVL.astAxes[stMasterAxis.nIndex].stConfig.afSlaveAxisRatio[GVL.iAxis] := nNO_GEARING;
            FOR nSlaveAxesIndex := 1 TO GVL_APP.nAXIS_NUM DO
                GVL.astAxes[nSlaveAxesIndex].stConfig.afMultiSlaveAxisRatio[GVL.iAxis] := nNO_GEARING;
            END_FOR
        END_IF

    E_MotionFunctions.eHome:
        fbHome.bExecute := stAxisStruct.stControl.bExecute AND NOT stAxisStruct.stStatus.bError;
        fbHome.eHomeSeq := stAxisStruct.stConfig.eHomeSeq;
        fbHome.fHomePosition := stAxisStruct.stConfig.fHomePosition;
        fbHome.fHomeFinishDistance := stAxisStruct.stConfig.fHomeFinishDistance;
        bDoneEdge := fbHome.bDone;
        bCommandAbortedEdge := fbHome.bCommandAborted;

    E_MotionFunctions.eWriteParameter:
        fbWriteParameter.Execute := stAxisStruct.stcontrol.bExecute;
        fbWriteParameter.ParameterNumber := stAxisStruct.stConfig.eAxisParameters;
        fbWriteParameter.Value := stAxisStruct.stConfig.fWriteAxisParameter;
        bDoneEdge := fbWriteParameter.Done;

END_CASE

//Busy from the motion function blocks
stAxisStruct.stStatus.bBusy := bBusy;

//CommandAborted from the eCommand function blocks
fbCommandAbortedRiseEdge(CLK:= bCommandAbortedEdge);
IF fbCommandAbortedRiseEdge.Q THEN
    stAxisStruct.stStatus.bCommandAborted := TRUE;
END_IF

//Done from the eCommand function blocks
fbDoneRiseEdge(CLK:= bDoneEdge);
IF fbDoneRiseEdge.Q THEN
    stAxisStruct.stStatus.bDone := TRUE;
    stAxisStruct.stStatus.bCommandAborted:=FALSE;
END_IF

//Reset Done and CommandAborted with any new eCommand (Execute or Jog)
fbExecuteRiseEdge(CLK:=stAxisStruct.stControl.bExecute);
IF fbExecuteRiseEdge.Q THEN
    stAxisStruct.stStatus.bDone := FALSE;
    stAxisStruct.stStatus.bCommandAborted := FALSE;
END_IF
fbJogRiseEdge(CLK:=stAxisStruct.stControl.bJogBwd OR stAxisStruct.stControl.bJogFwd);
IF fbJogRiseEdge.Q AND (stAxisStruct.stControl.eCommand = E_MotionFunctions.eJog) THEN
    stAxisStruct.stStatus.bDone := FALSE;
    stAxisStruct.stStatus.bCommandAborted := FALSE;
END_IF

//Execution of fbReset ended
fbResetFinishedRiseEdge(CLK:=fbReset.Done OR fbReset.Error);
IF fbResetFinishedRiseEdge.Q THEN
    stAxisStruct.stControl.bReset := FALSE;
    IF NOT fbReset.Error THEN
        stAxisStruct.stStatus.bError := FALSE;
        stAxisStruct.stStatus.nErrorID := 0;
        stAxisStruct.stError.nResetErrorID := 0;
    END_IF
    stAxisStruct.stError.nNCErrorID := 0;
    stAxisStruct.stError.nGearInErrorID := 0;
    stAxisStruct.stError.nGearInMultiMasterErrorID := 0;
    stAxisStruct.stError.nGearOutErrorID := 0;
    stAxisStruct.stError.fbReadParameterErrorId := 0;
    stAxisStruct.stError.fbWriteParameterErrorId := 0;
    stAxisStruct.stError.nPowerErrorID := 0;
    stAxisStruct.stError.nStopErrorID := 0;
    stAxisStruct.stError.nHaltErrorID := 0;
    stAxisStruct.stError.nHomeErrorID := 0;
    stAxisStruct.stError.nJogErrorID := 0;
    stAxisStruct.stError.nMoveAbsoluteErrorID := 0;
    stAxisStruct.stError.nMoveRelativeErrorID := 0;
    stAxisStruct.stError.nMoveModuloErrorID := 0;
    stAxisStruct.stError.nMoveVelocityErrorID := 0;
    stAxisStruct.stControl.bExecute := FALSE;
    stAxisStruct.stControl.bStop := FALSE;
    stAxisStruct.stControl.bHalt := FALSE;
    stAxisStruct.stControl.bJogBwd := FALSE;
    stAxisStruct.stControl.bJogFwd := FALSE;
END_IF

//Execution of fbStop ended
fbStopFinishedRiseEdge(CLK:=fbStop.Done OR fbStop.Error OR fbStop.CommandAborted);
IF fbStopFinishedRiseEdge.Q THEN
    stAxisStruct.stControl.bStop := FALSE;
END_IF

//Execution of fbHalt ended
fbHaltFinishedRiseEdge(CLK:=fbHalt.Done OR fbHalt.Error OR fbHalt.CommandAborted);
IF fbHaltFinishedRiseEdge.Q THEN
    stAxisStruct.stControl.bHalt := FALSE;
END_IF

//Save the errors from the PLCopen motion functions blocks and from the NC
IF fbPower.Error THEN
    stAxisStruct.stStatus.bError := TRUE;
    stAxisStruct.stStatus.nErrorId := fbPower.ErrorID;
    stAxisStruct.stError.nPowerErrorID := fbPower.ErrorID;

ELSIF fbHalt.Error THEN
    stAxisStruct.stStatus.bError := TRUE;
    stAxisStruct.stStatus.nErrorId := fbHalt.ErrorID;
    stAxisStruct.stError.nHaltErrorID := fbHalt.ErrorID;

ELSIF fbStop.Error THEN
    stAxisStruct.stStatus.bError := TRUE;
    stAxisStruct.stStatus.nErrorId := fbStop.ErrorID;
    stAxisStruct.stError.nStopErrorID := fbStop.ErrorID;

ELSIF fbHalt.Error THEN
    stAxisStruct.stStatus.bError := TRUE;
    stAxisStruct.stStatus.nErrorId := fbHalt.ErrorID;
    stAxisStruct.stError.nHaltErrorID := fbHalt.ErrorID;

ELSIF fbReset.Error THEN
    stAxisStruct.stStatus.bError := TRUE;
    stAxisStruct.stStatus.nErrorId := fbReset.ErrorID;
    stAxisStruct.stError.nResetErrorID := fbReset.ErrorID;

ELSIF fbJog.Error THEN
    stAxisStruct.stStatus.bError := TRUE;
    stAxisStruct.stStatus.nErrorId := fbJog.ErrorID;
    stAxisStruct.stError.nJogErrorID := fbJog.ErrorID;

ELSIF fbMoveVelocity.Error THEN
    stAxisStruct.stStatus.bError := TRUE;
    stAxisStruct.stStatus.nErrorId := fbMoveVelocity.ErrorID;
    stAxisStruct.stError.nMoveVelocityErrorID := fbMoveVelocity.ErrorID;

ELSIF fbMoveRelative.Error THEN
    stAxisStruct.stStatus.bError := TRUE;
    stAxisStruct.stStatus.nErrorId := fbMoveRelative.ErrorID;
    stAxisStruct.stError.nMoveRelativeErrorID := fbMoveRelative.ErrorID;

ELSIF fbMoveAbsolute.Error THEN
    stAxisStruct.stStatus.bError := TRUE;
    stAxisStruct.stStatus.nErrorId := fbMoveAbsolute.ErrorID;
    stAxisStruct.stError.nMoveAbsoluteErrorID := fbMoveAbsolute.ErrorID;

ELSIF fbMoveModulo.Error THEN
    stAxisStruct.stStatus.bError := TRUE;
    stAxisStruct.stStatus.nErrorId := fbMoveModulo.ErrorID;
    stAxisStruct.stError.nMoveModuloErrorID := fbMoveModulo.ErrorID;

ELSIF fbHome.bError THEN
    stAxisStruct.stStatus.bError := TRUE;
    stAxisStruct.stStatus.nErrorId := fbHome.nErrorID;
    stAxisStruct.stError.nHomeErrorID := fbHome.nErrorID;

ELSIF fbGearIn.Error THEN
    stAxisStruct.stStatus.bError := TRUE;
    stAxisStruct.stStatus.nErrorId := fbGearIn.ErrorID;
    stAxisStruct.stError.nGearInErrorId:=fbGearIn.ErrorID;

ELSIF fbGearInMultiMaster.Error THEN
    stAxisStruct.stStatus.bError := TRUE;
    stAxisStruct.stStatus.nErrorId:=fbGearInMultiMaster.ErrorID;
    stAxisStruct.stError.nGearInMultiMasterErrorId:=fbGearInMultiMaster.ErrorID;

ELSIF fbGearOut.Error and stAxisStruct.Axis.Status.Coupled THEN
    stAxisStruct.stStatus.bError := TRUE;
    stAxisStruct.stStatus.nErrorId := fbGearOut.ErrorID;
    stAxisStruct.stError.nGearOutErrorId := fbGearOut.ErrorID;

ELSIF fbWriteParameter.Error THEN
    stAxisStruct.stStatus.bError := TRUE;
    stAxisStruct.stStatus.nErrorId := fbWriteParameter.ErrorID;
    stAxisStruct.stError.fbWriteParameterErrorId := fbWriteParameter.ErrorID;

ELSIF fbReadParameter.Error THEN
    stAxisStruct.stStatus.bError := TRUE;
    stAxisStruct.stStatus.nErrorId := fbReadParameter.ErrorID;
    stAxisStruct.stError.fbReadParameterErrorId:=fbReadParameter.ErrorID;

ELSIF stAxisStruct.Axis.Status.Error THEN
    stAxisStruct.stStatus.bError := stAxisStruct.Axis.Status.Error;
    stAxisStruct.stStatus.nErrorId := stAxisStruct.Axis.Status.ErrorID;
    stAxisStruct.stError.nNCErrorId := stAxisStruct.Axis.Status.ErrorID;

END_IF;

//Actual Velocity
stAxisStruct.stStatus.fActVelocity := stAxisStruct.Axis.NcToPlc.ActVelo;

//Actual Position
IF stAxisStruct.Axis.Status.OpMode.Modulo THEN
    stAxisStruct.stStatus.fActPosition := stAxisStruct.Axis.NcToPlc.ModuloActPos;
ELSE
    stAxisStruct.stStatus.fActPosition := stAxisStruct.Axis.NcToPlc.ActPos;
END_IF

//Homing status
stAxisStruct.stStatus.bHomed := stAxisStruct.Axis.Status.Homed;

//Moving Status from the NC
stAxisStruct.stStatus.bMoving := stAxisStruct.Axis.Status.Moving;

//Gearing Status from the NC
stAxisStruct.stStatus.bGeared := stAxisStruct.Axis.Status.Coupled;

IF stAxisStruct.Axis.Status.Coupled AND stAxisStruct.Axis.PlcToNc.GearRatio1 <> 0 AND stAxisStruct.stConfig.astMultiMasterAxisLatched[1].nIndex <> 0 THEN
    GVL.astAxes[stAxisStruct.stConfig.astMultiMasterAxisLatched[1].nIndex].stConfig.afMultiSlaveAxisRatio[GVL.iAxis] := stAxisStruct.Axis.PlcToNc.GearRatio1;
    stAxisStruct.stStatus.bCoupledGear1 := TRUE;
ELSE
    stAxisStruct.stStatus.bCoupledGear1 := FALSE;
END_IF

IF stAxisStruct.Axis.Status.Coupled AND stAxisStruct.Axis.PlcToNc.GearRatio2 <> 0 AND stAxisStruct.stConfig.astMultiMasterAxisLatched[2].nIndex <> 0 THEN
    GVL.astAxes[stAxisStruct.stConfig.astMultiMasterAxisLatched[2].nIndex].stConfig.afMultiSlaveAxisRatio[GVL.iAxis] := stAxisStruct.Axis.PlcToNc.GearRatio2;
    stAxisStruct.stStatus.bCoupledGear2 := TRUE;
ELSE
    stAxisStruct.stStatus.bCoupledGear2 := FALSE;
END_IF

IF stAxisStruct.Axis.Status.Coupled AND stAxisStruct.Axis.PlcToNc.GearRatio3 <> 0 AND stAxisStruct.stConfig.astMultiMasterAxisLatched[3].nIndex <> 0 THEN
    GVL.astAxes[stAxisStruct.stConfig.astMultiMasterAxisLatched[3].nIndex].stConfig.afMultiSlaveAxisRatio[GVL.iAxis] := stAxisStruct.Axis.PlcToNc.GearRatio3;
    stAxisStruct.stStatus.bCoupledGear3 := TRUE;
ELSE
    stAxisStruct.stStatus.bCoupledGear3 := FALSE;
END_IF

IF stAxisStruct.Axis.Status.Coupled AND stAxisStruct.Axis.PlcToNc.GearRatio4 <> 0 AND stAxisStruct.stConfig.astMultiMasterAxisLatched[4].nIndex <> 0 THEN
    GVL.astAxes[stAxisStruct.stConfig.astMultiMasterAxisLatched[4].nIndex].stConfig.afMultiSlaveAxisRatio[GVL.iAxis] := stAxisStruct.Axis.PlcToNc.GearRatio4;
    stAxisStruct.stStatus.bCoupledGear4 := TRUE;
ELSE
    stAxisStruct.stStatus.bCoupledGear4 := FALSE;
END_IF

//Reset bExecute
stAxisStruct.stControl.bExecute := FALSE;

ACTION actReadMcParameters:
(*This act reads the MC parameters using an MC_ReadParameter FB FOR each variable
Intended TO be executed once every PLC cycle
Another FB is used TO trasnfer default axis parameters TO the stAxisStruct so
bReadValid is used TO halt that trasnfer UNTIL the parameters have been
read successfully. It may take a couple OF cycles once the PLC starts up.*)

//Slow jogging Velocity
fbReadAxisVeloManSlow(Axis := stAxisStruct.Axis,
                        Enable:= TRUE,
                        ReadMode:= READMODE_CYCLIC,
                        ParameterNumber := E_AxisParameters.AxisManualVelocitySlow,
                        Value=> stAxisStruct.stConfig.fVelocityDefaultSlow);
//Fast jogging velocity
fbReadAxisVeloManFast(Axis := stAxisStruct.Axis,
                        Enable:= TRUE,
                        ReadMode:= READMODE_CYCLIC,
                        ParameterNumber := E_AxisParameters.AxisManualVelocityFast,
                        Value=> stAxisStruct.stConfig.fVelocityDefaultFast);
//Homing velocity to Cam
fbReadHomingVelToCam(Axis := stAxisStruct.Axis,
                        Enable:= TRUE,
                        ReadMode:= READMODE_CYCLIC,
                        ParameterNumber := E_AxisParameters.AxisVelocityToCam,
                        Value=> stAxisStruct.stConfig.fHomingVelToCam);
//Homing velocity from Cam
fbReadHomingVelFromCam(Axis := stAxisStruct.Axis,
                        Enable:= TRUE,
                        ReadMode:= READMODE_CYCLIC,
                        ParameterNumber := E_AxisParameters.AxisVelocityFromCam,
                        Value=> stAxisStruct.stConfig.fHomingVelFromCam);
//Max velocity
fbReadAxisVeloMax(Axis := stAxisStruct.Axis,
                        Enable:= TRUE,
                        ReadMode:= READMODE_CYCLIC,
                        ParameterNumber := E_AxisParameters.AxisMaxVelocity,
                        Value=> stAxisStruct.stConfig.fVeloMax);
//Acceleration
fbReadAxisAcc(Axis := stAxisStruct.Axis,
                        Enable:= TRUE,
                        ReadMode:= READMODE_CYCLIC,
                        ParameterNumber := E_AxisParameters.AxisAccMax,
                        Value=> stAxisStruct.stConfig.fDefaultAcc);
//Deceleration
fbReadAxisDec(Axis := stAxisStruct.Axis,
                        Enable:= TRUE,
                        ReadMode:= READMODE_CYCLIC,
                        ParameterNumber := E_AxisParameters.AxisDecMax,
                        Value=> stAxisStruct.stConfig.fDefaultDec);

//Soft limits enabled
fbReadEnMinSoftPosLimit(Axis := stAxisStruct.Axis,
                        Enable:= TRUE,
                        ReadMode:= READMODE_CYCLIC,
                        ParameterNumber := E_AxisParameters.EnableLimitBackward);
stAxisStruct.stConfig.bEnMinSoftPosLimit:= LREAL_TO_BOOL(fbReadEnMinSoftPosLimit.Value);

fbReadEnMaxSoftPosLimit(Axis := stAxisStruct.Axis,
                        Enable:= TRUE,
                        ReadMode:= READMODE_CYCLIC,
                        ParameterNumber := E_AxisParameters.EnableLimitForward);
stAxisStruct.stConfig.bEnMaxSoftPosLimit:= LREAL_TO_BOOL(fbReadEnMaxSoftPosLimit.Value);

//Soft limit values
fbReadMinSoftPosLimit(Axis := stAxisStruct.Axis,
                        Enable:= TRUE,
                        ReadMode:= READMODE_CYCLIC,
                        ParameterNumber := E_AxisParameters.SWLimitBackward,
                        Value=>stAxisStruct.stConfig.fMinSoftPosLimit);
fbReadMaxSoftPosLimit(Axis := stAxisStruct.Axis,
                        Enable:= TRUE,
                        ReadMode:= READMODE_CYCLIC,
                        ParameterNumber := E_AxisParameters.SWLimitForward,
                        Value=>stAxisStruct.stConfig.fMaxSoftPosLimit);

//Position Lag Monitoring
fbReadEnPositionLagMonitoring(Axis := stAxisStruct.Axis,
                        Enable:= TRUE,
                        ReadMode:= READMODE_CYCLIC,
                        ParameterNumber := E_AxisParameters.EnablePositionLagMonitoring);
stAxisStruct.stConfig.bEnPositionLagMonitoring:= LREAL_TO_BOOL(fbReadEnPositionLagMonitoring.Value);

fbReadAxisMaxPosLagValue(Axis := stAxisStruct.Axis,
                        Enable:= TRUE,
                        ReadMode:= READMODE_CYCLIC,
                        ParameterNumber := E_AxisParameters.MaxPositionLag,
                        Value=>stAxisStruct.stConfig.fMaxPosLagValue);

// Target Position Monitoring
fbReadEnTargetPositionMonitoring(Axis := stAxisStruct.Axis,
                        Enable:= TRUE,
                        ReadMode:= READMODE_CYCLIC,
                        ParameterNumber := E_AxisParameters.SWLimitBackward);
stAxisStruct.stConfig.bEnTargetPositionMonitoring:= LREAL_TO_BOOL(fbReadEnTargetPositionMonitoring.Value);

fbReadTargetPositionWindow(Axis := stAxisStruct.Axis,
                        Enable:= TRUE,
                        ReadMode:= READMODE_CYCLIC,
                        ParameterNumber := E_AxisParameters.AxisTargetPositionWindow,
                        Value=> stAxisStruct.stConfig.fTargetPositionWindow);

//All variables are valid
stAxisStruct.stConfig.bReadMcParametersValid:= FALSE;
stAxisStruct.stConfig.bReadMcParametersValid:= fbReadAxisVeloManSlow.Valid AND
    fbReadAxisVeloManFast.Valid AND
    fbReadHomingVelToCam.Valid AND
    fbReadHomingVelFromCam.Valid AND
    fbReadAxisVeloMax.Valid AND
    fbReadAxisAcc.Valid AND
    fbReadAxisDec.Valid AND
    fbReadEnMinSoftPosLimit.Valid AND
    fbReadEnMaxSoftPosLimit.Valid AND
    fbReadMinSoftPosLimit.Valid AND
    fbReadMaxSoftPosLimit.Valid AND
    fbReadEnPositionLagMonitoring.Valid AND
    fbReadAxisMaxPosLagValue.Valid AND
    fbReadEnTargetPositionMonitoring.Valid AND
    fbReadTargetPositionWindow.Valid;

//One of the variables has a read error
stAxisStruct.stConfig.bReadMcParametersError:= fbReadAxisVeloManSlow.Error OR
    fbReadAxisVeloManFast.Error OR
    fbReadHomingVelToCam.Error OR
    fbReadHomingVelFromCam.Valid OR
    fbReadAxisVeloMax.Error OR
    fbReadAxisAcc.Error OR
    fbReadAxisDec.Error OR
    fbReadEnMinSoftPosLimit.Error OR
    fbReadEnMaxSoftPosLimit.Error OR
    fbReadMinSoftPosLimit.Error OR
    fbReadMaxSoftPosLimit.Error OR
    fbReadEnPositionLagMonitoring.Error OR
    fbReadAxisMaxPosLagValue.Error OR
    fbReadEnTargetPositionMonitoring.Error OR
    fbReadTargetPositionWindow.Error;
END_ACTION

END_FUNCTION_BLOCK

// ---- POUs/Motion/Homing/FB_Homing.TcPOU
FUNCTION_BLOCK FB_Homing
VAR_IN_OUT
    Axis: Axis_Ref;
END_VAR
VAR_INPUT
    bExecute: BOOL;
    bLimitFwd: BOOL;
    bLimitBwd: BOOL;
    bHomeSensor: BOOL;
    eHomeSeq: E_HomingRoutines;
    fHomePosition: LREAL;
    fHomeFinishDistance: LREAL;
END_VAR
VAR_OUTPUT
    bDone : BOOL;
    bBusy: BOOL;
    bCommandAborted: BOOL;
    bError: BOOL;
    nErrorId: UDINT;
END_VAR
VAR
    //Beckhoff homing function blocks
    fbStepLimitSwitchPreparation: MC_StepLimitSwitchDetection;
    fbStepLimitSwitchDetection: MC_StepLimitSwitchDetection;
    fbStepAbsoluteSwitchDetection: MC_StepAbsoluteSwitchDetection;
    fbStepReferencePulseDetection: MC_StepReferencePulseDetection;
    fbHomeDirect: MC_HomeDirect;
    fbSetPos: MC_SetPosition;
    fbFinishHoming: MC_FinishHoming;
    fbAbortHoming: MC_AbortHoming;
    //Hardware Signals
    eLimitSwitchMode: MC_Switch_Mode := mcRisingEdge;
    stLimitSwitchSignal: MC_Ref_Signal_Ref;
    eRefSwitchMode: MC_Switch_Mode := mcRisingEdge;
    stRefSwitchSignal: MC_Ref_Signal_Ref;
    stEncPulseSignal: MC_Ref_Signal_Ref;
    //Homing parameters
    stPreparationDirection: MC_Home_Direction;
    stDetectDirection: MC_Home_Direction;
    stHomingParameter: MC_HomingParameter;
    stOptions: ST_Home_Options4;
    fbVelocityToCam: MC_ReadParameter;
    fVelocityToCam: LREAL;
    fbVelocityFromCam: MC_ReadParameter;
    fVelocityFromCam: LREAL;
    //State machine
    fbExecute: R_TRIG;
    bViaLimitSwitch: BOOL;
    eHomingState: (eWaitForRequest := 0, ePreparation := 1, eDetection := 2, eSetPos := 3, eFinishHoming := 4, eAbortHoming := 20);
    iErrorId: UDINT;
    bDetectionFB_Execute: BOOL;
    bDetectionFB_Done: BOOL;
    bDetectionFB_Busy: BOOL;
    bDetectionFB_CommandAborted: BOOL;
    bDetectionFB_Error: BOOL;
    nDetectionFB_ErrorID: UDINT;
    fRecordedPosition: LREAL;
    fRecordedPositionLatched: LREAL;
END_VAR


//Hardware signals
stLimitSwitchSignal.SignalSource := SignalSource_Default;
stLimitSwitchSignal.TouchProbe := PlcEvent;
stRefSwitchSignal.SignalSource := SignalSource_Default;
stRefSwitchSignal.TouchProbe := PlcEvent;
stRefSwitchSignal.Level := bHomeSensor;
stEncPulseSignal.SignalSource := SignalSource_ZeroPulse;
stEncPulseSignal.TouchProbe := TouchProbe1;

//Constantly read the NC for homing velocities so they are available when a homing is executed
fbVelocityToCam(
    Axis := Axis,
    Enable := TRUE,
    ParameterNumber := E_AxisParameters.AxisVelocityToCam,
    ReadMode := READMODE_CYCLIC);

fbVelocityFromCam(
    Axis := Axis,
    Enable := TRUE,
    ParameterNumber := E_AxisParameters.AxisVelocityFromCam,
    ReadMode := READMODE_CYCLIC);

    //Only write velocity if the function block has not errored
IF NOT fbVelocityToCam.Error THEN
    fVelocityToCam := fbVelocityToCam.Value;
END_IF

IF NOT fbVelocityFromCam.Error THEN
    fVelocityFromCam := fbVelocityFromCam.Value;
END_IF

    //Feeds function block errors through
IF fbVelocityToCam.Error THEN
    bError := TRUE;
    nErrorID := fbVelocityToCam.ErrorID;

ELSIF fbVelocityFromCam.Error THEN
    bError := TRUE;
    nErrorID := fbVelocityFromCam.ErrorID;
END_IF

//Common function blocks used for all routines
stOptions.DisableDriveAccess:=TRUE;

fbStepLimitSwitchPreparation.Options.DisableDriveAccess := stOptions.DisableDriveAccess;
fbStepLimitSwitchPreparation(
    Axis := Axis,
    Parameter := stHomingParameter,
    Direction := stPreparationDirection,
    LimitSwitchMode:= eLimitSwitchMode,
    LimitSwitchSignal:= stLimitSwitchSignal,
    Velocity := fVelocityToCam);

fbSetPos(
    Axis := Axis,
    Position := Axis.NcToPlc.ActPos - fRecordedPositionLatched + fHomePosition);

fbFinishHoming.Options.DisableDriveAccess := stOptions.DisableDriveAccess;
fbFinishHoming(
    Axis := Axis,
    Parameter := stHomingParameter,
    Velocity := fVelocityFromCam);

fbAbortHoming.Options.DisableDriveAccess := stOptions.DisableDriveAccess;
fbAbortHoming(
    Axis := Axis,
    Parameter := stHomingParameter);

//ACTs contain function blocks custom to each individual routine for the detection stage
CASE eHomeSeq OF
    E_HomingRoutines.eHomeToLimit_Bwd,
    E_HomingRoutines.eHomeToLimit_Fwd:
        actHomeToLimit();

    E_HomingRoutines.eHomeToRef_Bwd,
    E_HomingRoutines.eHomeToRef_Fwd:
        actHomeToRef();

    E_HomingRoutines.eHomeToEncPulse_Bwd,
    E_HomingRoutines.eHomeToEncPulse_Fwd,
    E_HomingRoutines.eHomeToEncPulse_viaBwdLimit,
    E_HomingRoutines.eHomeToEncPulse_viaFwdLimit:
        actHomeToEncPulse();

    E_HomingRoutines.eHomeDirect:
        actHomeDirect();
END_CASE


//State machine
fbExecute(CLK:= bExecute);
CASE eHomingState OF

    eWaitForRequest:
        IF NOT bExecute THEN
            bBusy := FALSE;
            bDone := FALSE;
            bCommandAborted := FALSE;
            bError := FALSE;
            nErrorID := 0;
            iErrorID := 0;

            fbStepLimitSwitchPreparation.Execute := FALSE;
            fbStepLimitSwitchDetection.Execute := FALSE;
            fbStepAbsoluteSwitchDetection.Execute := FALSE;
            fbStepReferencePulseDetection.Execute := FALSE;
            fbHomeDirect.Execute := FALSE;
            fbSetPos.Execute := FALSE;
            fbFinishHoming.Execute := FALSE;
            fbAbortHoming.Execute := FALSE;
        END_IF

        IF fbExecute.Q THEN
            bBusy:= TRUE;
            eHomingState:= ePreparation;
        END_IF


    ePreparation: //If bViaLimitSwitch is set TRUE then go first to a limit otherwise skip this step
        IF bViaLimitSwitch THEN
            fbStepLimitSwitchPreparation.Execute := TRUE;
        ELSE
            eHomingState := eDetection;
        END_IF

        IF NOT fbStepLimitSwitchPreparation.Busy AND fbStepLimitSwitchPreparation.Done THEN
            fbStepLimitSwitchPreparation.Execute := FALSE;
            eHomingState := eDetection;
        ELSIF NOT fbStepLimitSwitchPreparation.Busy AND (fbStepLimitSwitchPreparation.Error OR fbStepLimitSwitchPreparation.CommandAborted) THEN
            iErrorID := fbStepLimitSwitchPreparation.ErrorID;
            fbStepLimitSwitchPreparation.Execute := FALSE;
            eHomingState := eAbortHoming;
        END_IF


    eDetection: //Use bDetectionFB_<BOOL Variables> to interact with different detection FBs located in ACTs
        bDetectionFB_Execute := TRUE;

        IF NOT bDetectionFB_Busy AND bDetectionFB_Done THEN
            bDetectionFB_Execute := FALSE;
            fRecordedPositionLatched := fRecordedPosition;
            IF eHomeSeq = E_HomingRoutines.eHomeDirect THEN
                eHomingState := eWaitForRequest;
            ELSE
                eHomingState := eSetPos;
            END_IF
        ELSIF NOT bDetectionFB_Busy AND (bDetectionFB_Error OR bDetectionFB_CommandAborted) THEN
            iErrorID := nDetectionFB_ErrorID;
            bDetectionFB_Execute := FALSE;
            eHomingState := eAbortHoming;
        END_IF


    eSetPos:
        fbSetPos.Execute := TRUE;

        fbSetPos.Options.ClearPositionLag := TRUE;
        IF NOT fbSetPos.Busy AND fbSetPos.Done THEN
            fbSetPos.Execute := FALSE;
            eHomingState := eFinishHoming;
        ELSIF NOT fbSetPos.Busy AND fbSetPos.Error THEN
            iErrorID := fbSetPos.ErrorID;
            fbSetPos.Execute := FALSE;
            eHomingState := eAbortHoming;
        END_IF


    eFinishHoming:
        fbFinishHoming.Execute := TRUE;

        IF NOT fbFinishHoming.Busy AND fbFinishHoming.Done THEN
            bBusy := FALSE;
            bDone := TRUE;
            fbFinishHoming.Execute := FALSE;
            eHomingState := eWaitForRequest;
        ELSIF NOT fbFinishHoming.Busy AND (fbFinishHoming.Error OR fbFinishHoming.CommandAborted) THEN
            iErrorID := fbFinishHoming.ErrorID;
            fbFinishHoming.Execute := FALSE;
            eHomingState := eAbortHoming;
        END_IF


    eAbortHoming:
        fbAbortHoming.Execute := TRUE;

        IF NOT fbAbortHoming.Busy AND fbAbortHoming.Done THEN
            bBusy := FALSE;
            IF iErrorId <> 0 THEN
                bError := TRUE;
                nErrorId := iErrorId;
            ELSE
                bCommandAborted := TRUE;
            END_IF
            fbAbortHoming.Execute := FALSE;
            eHomingState := eWaitForRequest;
        ELSIF NOT fbAbortHoming.Busy AND fbAbortHoming.Error THEN
            bBusy := FALSE;
            bError := TRUE;
            nErrorID := fbAbortHoming.ErrorID;
            fbAbortHoming.Execute := FALSE;
            eHomingState := eWaitForRequest;
        END_IF

END_CASE

ACTION actHomeDirect:
bViaLimitSwitch := FALSE;

fbHomeDirect(
    Axis := Axis,
    Parameter := stHomingParameter,
    Execute := bDetectionFB_Execute,
    SetPosition := fHomePosition,
    Done => bDetectionFB_Done,
    Busy => bDetectionFB_Busy,
    CommandAborted => bDetectionFB_CommandAborted,
    Error => bDetectionFB_Error,
    ErrorID => nDetectionFB_ErrorID);
END_ACTION

ACTION actHomeToEncPulse:
CASE eHomeSeq OF
    E_HomingRoutines.eHomeToEncPulse_Bwd:
        stDetectDirection := mcNegativeDirection;
        fbFinishHoming.Distance := fHomeFinishDistance;
        bViaLimitSwitch := FALSE;
    E_HomingRoutines.eHomeToEncPulse_Fwd:
        stDetectDirection := mcPositiveDirection;
        fbFinishHoming.Distance := -fHomeFinishDistance;
        bViaLimitSwitch := FALSE;
    E_HomingRoutines.eHomeToEncPulse_viaBwdLimit:
        stDetectDirection := mcPositiveDirection;
        fbFinishHoming.Distance := fHomeFinishDistance;
        stPreparationDirection := mcNegativeDirection;
        stLimitSwitchSignal.Level := NOT(bLimitBwd);
        bViaLimitSwitch := TRUE;
    E_HomingRoutines.eHomeToEncPulse_viaFwdLimit:
        stDetectDirection := mcNegativeDirection;
        fbFinishHoming.Distance := -fHomeFinishDistance;
        stPreparationDirection := mcPositiveDirection;
        stLimitSwitchSignal.Level := NOT(bLimitFwd);
        bViaLimitSwitch := TRUE;
END_CASE

fbStepReferencePulseDetection.Options.DisableDriveAccess:= stOptions.DisableDriveAccess;
fbStepReferencePulseDetection(
    Axis := Axis,
    Execute := bDetectionFB_Execute,
    Parameter := stHomingParameter,
    Direction := stDetectDirection,
    ReferenceSignal := stEncPulseSignal,
    Velocity := fVelocityFromCam,
    Options := stOptions,
    Done => bDetectionFB_Done,
    Busy => bDetectionFB_Busy,
    CommandAborted => bDetectionFB_CommandAborted,
    Error => bDetectionFB_Error,
    ErrorID => nDetectionFB_ErrorID,
    RecordedPosition => fRecordedPosition);
END_ACTION

ACTION actHomeToLimit:
CASE eHomeSeq OF
    E_HomingRoutines.eHomeToLimit_Bwd:
        stLimitSwitchSignal.Level := NOT(bLimitBwd);
        stDetectDirection:= mcNegativeDirection;
        fbFinishHoming.Distance := fHomeFinishDistance;
    E_HomingRoutines.eHomeToLimit_Fwd:
        stLimitSwitchSignal.Level := NOT(bLimitFwd);
        stDetectDirection:= mcPositiveDirection;
        fbFinishHoming.Distance := -fHomeFinishDistance;
END_CASE
bViaLimitSwitch:=FALSE;

fbStepLimitSwitchDetection.Options.DisableDriveAccess:= stOptions.DisableDriveAccess;
fbStepLimitSwitchDetection(
    Axis := Axis,
    Execute := bDetectionFB_Execute,
    Parameter := stHomingParameter,
    Direction := stDetectDirection,
    LimitSwitchMode := eLimitSwitchMode,
    LimitSwitchSignal := stLimitSwitchSignal,
    Velocity := fVelocityFromCam,
    Options := stOptions,
    Done => bDetectionFB_Done,
    Busy => bDetectionFB_Busy,
    CommandAborted => bDetectionFB_CommandAborted,
    Error => bDetectionFB_Error,
    ErrorID => nDetectionFB_ErrorID,
    RecordedPosition => fRecordedPosition);
END_ACTION

ACTION actHomeToRef:
CASE eHomeSeq OF
    E_HomingRoutines.eHomeToRef_Bwd:
        stDetectDirection := mcNegativeDirection;
        fbFinishHoming.Distance := fHomeFinishDistance;
    E_HomingRoutines.eHomeToRef_Fwd:
        stDetectDirection := mcPositiveDirection;
        fbFinishHoming.Distance := -fHomeFinishDistance;
END_CASE
bViaLimitSwitch := FALSE;

fbStepAbsoluteSwitchDetection.Options.DisableDriveAccess := stOptions.DisableDriveAccess;
fbStepAbsoluteSwitchDetection(
    Axis := Axis,
    Execute := bDetectionFB_Execute,
    Parameter := stHomingParameter,
    Direction := stDetectDirection,
    SwitchMode := eRefSwitchMode,
    ReferenceSignal := stRefSwitchSignal,
    Velocity := fVelocityFromCam,
    PositiveLimitSwitch := NOT(bLimitFwd),
    NegativeLimitSwitch := NOT(bLimitBwd),
    Options := stOptions,
    Done => bDetectionFB_Done,
    Busy => bDetectionFB_Busy,
    CommandAborted => bDetectionFB_CommandAborted,
    Error => bDetectionFB_Error,
    ErrorID => nDetectionFB_ErrorID,
    RecordedPosition => fRecordedPosition);
END_ACTION

END_FUNCTION_BLOCK
